// Mitsubishi GX Works2 project: SOFI_AmitGitai[1]   PLC: FX3G

// global labels: Global1
VAR_GLOBAL
  CreamTank AT D1102 : INT;
  ChocolateTank AT D1110 : INT;
  BiscuitTank AT D1106 : INT;
END_VAR
VAR_GLOBAL CONSTANT
  SUBCream : INT := 300;
  SUBBiscuit : INT := 6;
END_VAR
VAR_GLOBAL
  TurnON AT X010 : BOOL;
  InventoryDownload AT X011 : BOOL;
  EmergencyOff AT X005 : BOOL;
  ZilufOn AT Y004 : BOOL;
  Sen_15 AT X004 : BOOL;
  Ariza AT X000 : BOOL;
  Sen_camera AT X002 : BOOL;
  Sen_contact AT X003 : BOOL;
  MachineAOn AT M0 : BOOL;
  TCoil1 AT TC1 : BOOL;
  Light1 AT Y001 : BOOL;
  TS1change AT TS1 : BOOL;
  RestartTimer AT M1 : BOOL;
  TS2change AT TS2 : BOOL;
  Light0 AT Y000 : BOOL;
  TCoil2 AT TC2 : BOOL;
  TCoil0 AT TC0 : BOOL;
  TS0change AT TS0 : BOOL;
  StartDgima AT X006 : BOOL;
  analog_input_1 AT D8280 : INT;
  save_analog_value AT D8000 : INT;
  HelperLight2 AT M2 : BOOL;
  StartDay AT X007 : BOOL;
  StartLamp AT Y007 : BOOL;
  Sen_30 AT X001 : BOOL;
END_VAR
VAR_GLOBAL CONSTANT
  MinimumChocolate : INT := 240;
END_VAR
VAR_GLOBAL
  CreamInput AT D1100 : INT;
  ChocolateInput AT D1108 : INT;
  BiscuitInput AT D1104 : INT;
  TCoil3 AT TC3 : BOOL;
  TS3Hivhuv AT TS3 : BOOL;
  HelperGoodInventory AT M4 : BOOL;
END_VAR
VAR_GLOBAL CONSTANT
  TimerHivHuv1 : INT := 6;
  TimerHivHuv2 : INT := 6;
END_VAR
VAR_GLOBAL
  ZilufTank AT D1112 : INT;
END_VAR
VAR_GLOBAL CONSTANT
  Hivhuv : INT := 30;
  RegularCoating : INT := 5;
  ChocolateAmountCoating : INT := 120;
  DoubleCoatingMinimum : INT := 6;
  DoubleCoatimgMaximum : INT := 10;
END_VAR
VAR_GLOBAL
  CoatingLamp AT Y003 : BOOL;
  TvilaTank AT D1116 : INT;
END_VAR
VAR_GLOBAL CONSTANT
  ChocolateAmountCoating2 : INT := 240;
END_VAR
VAR_GLOBAL
  TCoil4 AT TC4 : BOOL;
END_VAR
VAR_GLOBAL CONSTANT
  Timer50 : INT := 50;
  TimerFor4seconds : INT := 40;
  normal_chocolate : INT := 400;
END_VAR
VAR_GLOBAL
  ChocolateInputCoating AT D1118 : INT;
  TS4ForLamp AT TS4 : BOOL;
END_VAR
VAR_GLOBAL CONSTANT
  ResetTvilaTank : INT;
END_VAR
VAR_GLOBAL
  OutputC AT CS1 : BOOL;
  ArizaLamp AT Y002 : BOOL;
  InputC2 AT CC2 : BOOL;
END_VAR
VAR_GLOBAL CONSTANT
  Counter6 : INT := 6;
  Counter5 : INT := 5;
END_VAR
VAR_GLOBAL
  OutputC2 AT CS2 : BOOL;
  InputC AT CC1 : BOOL;
  FinishInputReciever AT M13 : BOOL;
  KrembosAmount AT D1120 : INT;
END_VAR
VAR_GLOBAL CONSTANT
  MishtahFinish : INT := 6;
END_VAR
VAR_GLOBAL
  analog_output AT D8282 : INT;
  STAM AT Y011 : BOOL;
END_VAR
VAR_GLOBAL CONSTANT
  CONST : INT;
END_VAR
VAR_GLOBAL
  KremboNew AT D1121 : INT;
END_VAR
VAR_GLOBAL CONSTANT
  const10 : INT := 10;
  CONST400 : INT := 400;
  CONST40 : INT := 40;
END_VAR
VAR_GLOBAL
  SubIndication AT M6 : BOOL;
  DgimaLamp AT M9 : BOOL;
  HelperLight3 AT M3 : BOOL;
  NoInventory AT M5 : BOOL;
  RegularCoat AT M7 : BOOL;
  DoubleCoat AT M8 : BOOL;
  ChocolateSubInventory AT M10 : BOOL;
  FinishZiluf AT M11 : BOOL;
  HelperM12 AT M12 : BOOL;
  HelperM15 AT M15 : BOOL;
  HelperM14 AT M14 : BOOL;
  HelperM16 AT M16 : BOOL;
  HelperM17 AT M17 : BOOL;
  HelperM18 AT M18 : BOOL;
  HelperM19 AT M19 : BOOL;
  HelperM20 AT M20 : BOOL;
  HelperM21 AT M21 : BOOL;
  HelperM22 AT M22 : BOOL;
  GoodInventory AT M24 : BOOL;
  HelperM25 AT M25 : BOOL;
  HelperM26 AT M26 : BOOL;
  HelperM27 AT M27 : BOOL;
  FinishDay AT M28 : BOOL;
  HelperM23 AT M23 : BOOL;
  HelperM29 AT M29 : BOOL;
  TCoil5 AT TC5 : BOOL;
  TS5Reset AT TS5 : BOOL;
END_VAR

// task Task_01 (event TRUE, interval 0, priority 31): POU_01

PROGRAM POU_01
VAR
  TS4 : BOOL;
  TSForLamp : BOOL;
END_VAR
(* structured ladder/FBD written out as ST: instructions are called as NAME(EN, inputs, outputs); _pN, _eN, _tN stand for wires *)
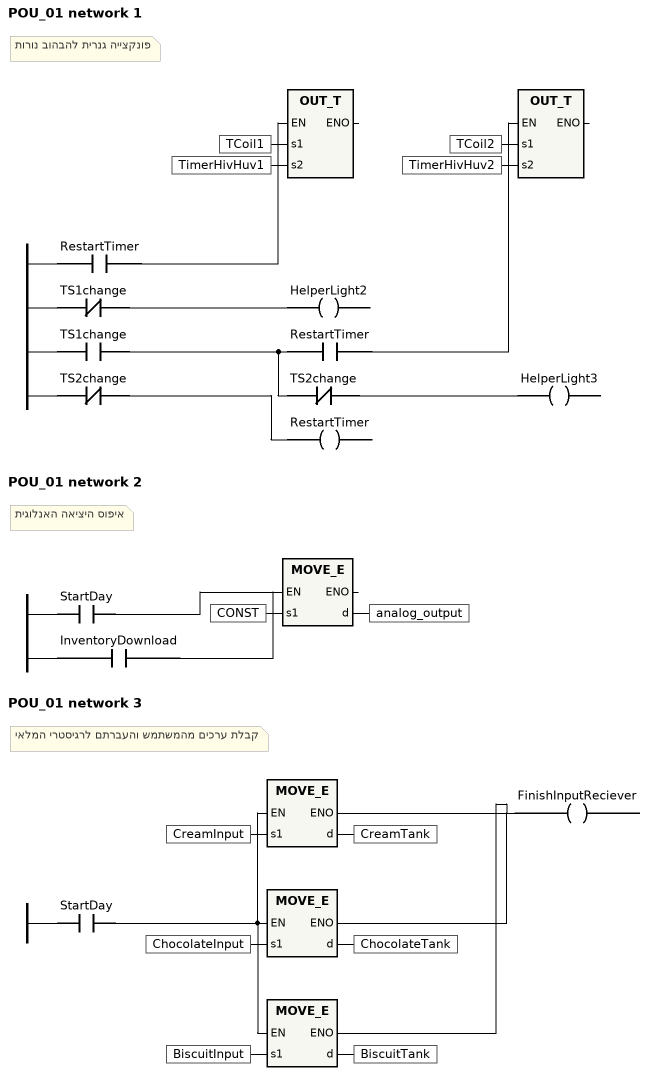
(* network 1 *)
(* פונקצייה גנרית להבהוב נורות *)
OUT_T(RestartTimer, TCoil1, TimerHivHuv1);
HelperLight2 := NOT TS1change;
OUT_T(TS1change AND RestartTimer, TCoil2, TimerHivHuv2);
HelperLight3 := TS1change AND NOT TS2change;
RestartTimer := NOT TS2change;
(* network 2 *)
(* איפוס היציאה האנלוגית *)
MOVE_E(StartDay OR InventoryDownload, CONST, analog_output);
(* network 3 *)
(* קבלת ערכים מהמשתמש והעברתם לרגיסטרי המלאי *)
_e1 := MOVE_E(StartDay, CreamInput, CreamTank);
_e2 := MOVE_E(StartDay, ChocolateInput, ChocolateTank);
_e3 := MOVE_E(StartDay, BiscuitInput, BiscuitTank);
FinishInputReciever := _e1 OR _e2 OR _e3;
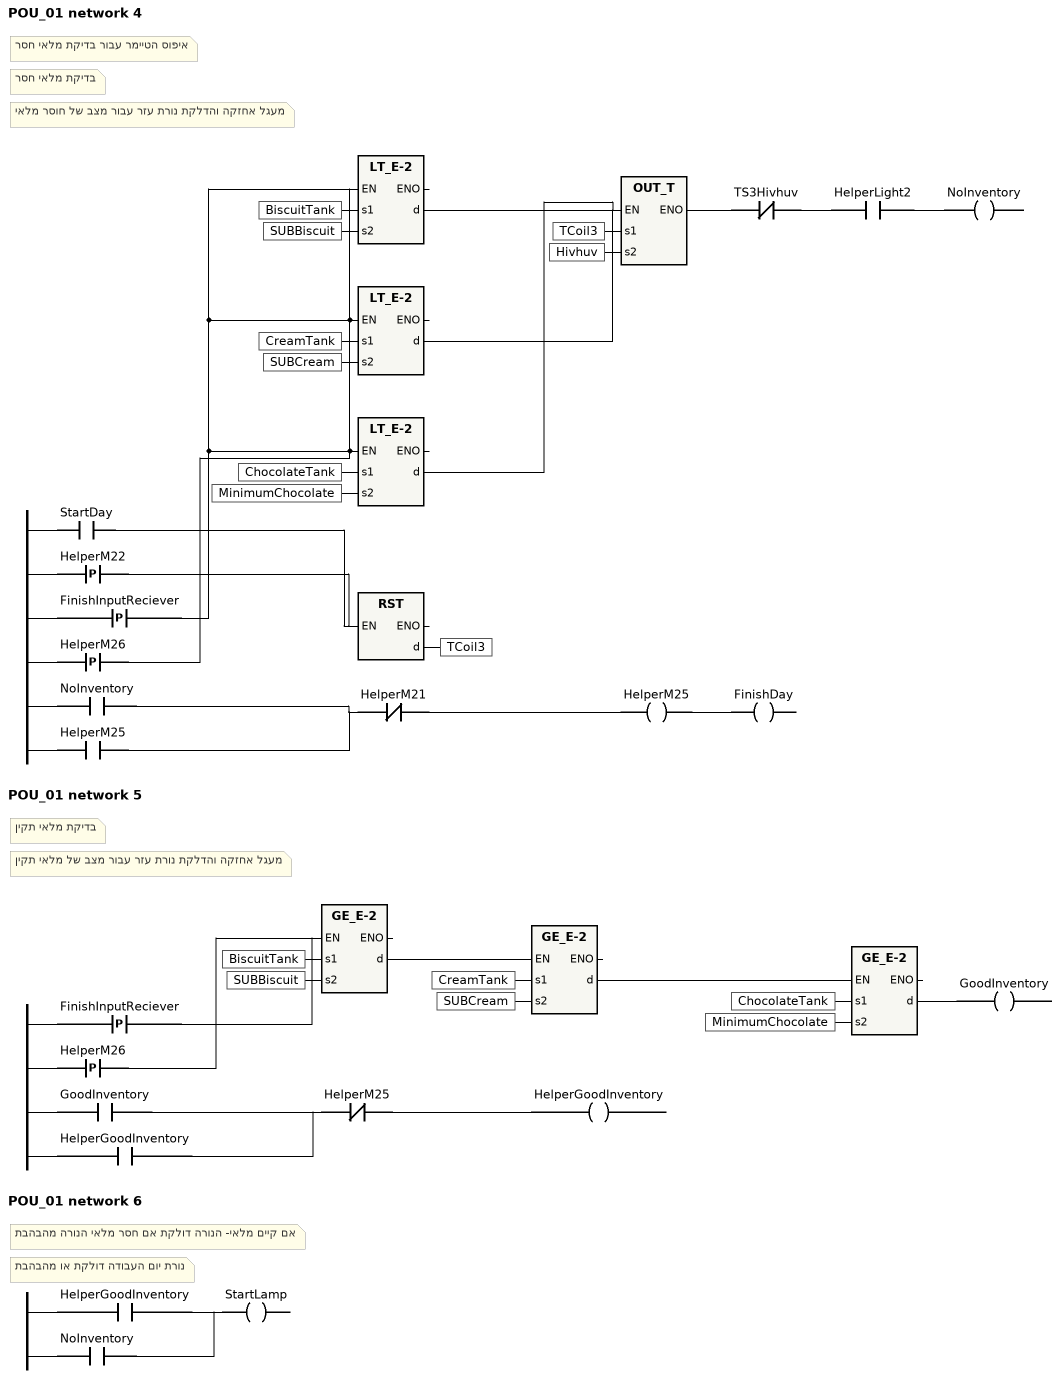
(* network 4 *)
(* איפוס הטיימר עבור בדיקת מלאי חסר *)
(* בדיקת מלאי חסר *)
(* מעגל אחזקה והדלקת נורת עזר עבור מצב של חוסר מלאי *)
RST(StartDay OR LDP(TRUE, HelperM22), TCoil3);
_p1 := LDP(TRUE, FinishInputReciever) OR LDP(TRUE, HelperM26);
LT_E(_p1, BiscuitTank, SUBBiscuit, _t2);
LT_E(_p1, CreamTank, SUBCream, _t3);
LT_E(_p1, ChocolateTank, MinimumChocolate, _t4);
_e5 := OUT_T(_t2 OR _t3 OR _t4, TCoil3, Hivhuv);
NoInventory := _e5 AND NOT TS3Hivhuv AND HelperLight2;
_p6 := (NoInventory OR HelperM25) AND NOT HelperM21;
HelperM25 := _p6;
FinishDay := _p6;
(* network 5 *)
(* בדיקת מלאי תקין *)
(* מעגל אחזקה והדלקת נורת עזר עבור מצב של מלאי תקין *)
GE_E(LDP(TRUE, FinishInputReciever) OR LDP(TRUE, HelperM26), BiscuitTank, SUBBiscuit, _t1);
GE_E(_t1, CreamTank, SUBCream, _t2);
GE_E(_t2, ChocolateTank, MinimumChocolate, _t3);
GoodInventory := _t3;
HelperGoodInventory := (GoodInventory OR HelperGoodInventory) AND NOT HelperM25;
(* network 6 *)
(* אם קיים מלאי- הנורה דולקת אם חסר מלאי הנורה מהבהבת *)
(* נורת יום העבודה דולקת או מהבהבת *)
StartLamp := HelperGoodInventory OR NoInventory;
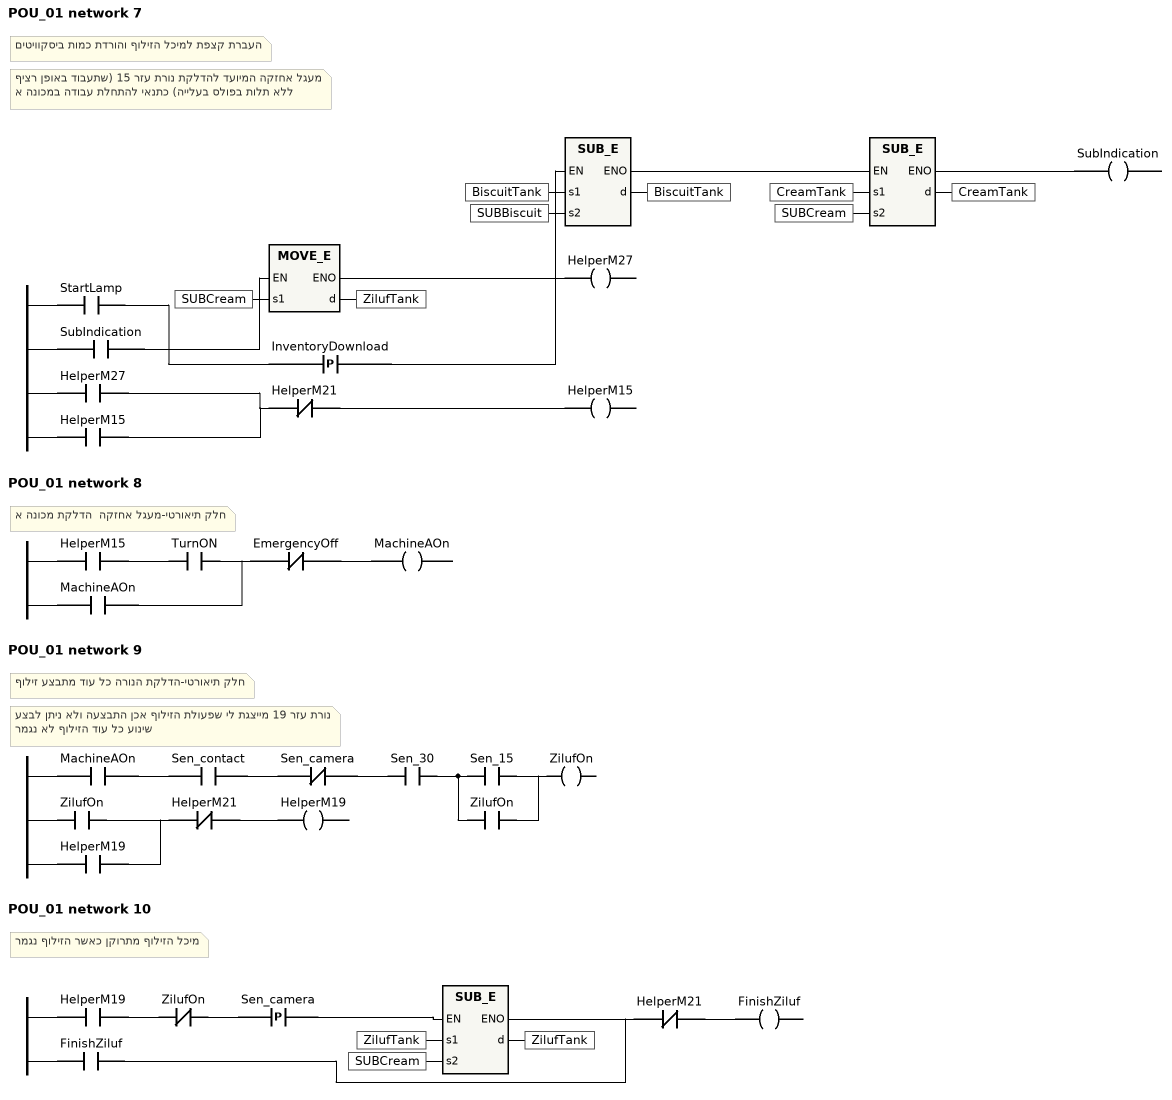
(* network 7 *)
(* העברת קצפת למיכל הזילוף והורדת כמות ביסקוויטים *)
(* מעגל אחזקה המיועד להדלקת נורת עזר 15 (שתעבוד באופן רציף ללא תלות בפולס בעלייה) כתנאי להתחלת עבודה במכונה א *)
_e1 := SUB_E(StartLamp AND LDP(TRUE, InventoryDownload), BiscuitTank, SUBBiscuit, BiscuitTank);
_e2 := SUB_E(_e1, CreamTank, SUBCream, CreamTank);
SubIndication := _e2;
_e3 := MOVE_E(SubIndication, SUBCream, ZilufTank);
HelperM27 := _e3;
HelperM15 := (HelperM27 OR HelperM15) AND NOT HelperM21;
(* network 8 *)
(* חלק תיאורטי-מעגל אחזקה  הדלקת מכונה א *)
MachineAOn := ((HelperM15 AND TurnON) OR MachineAOn) AND NOT EmergencyOff;
(* network 9 *)
(* חלק תיאורטי-הדלקת הנורה כל עוד מתבצע זילוף *)
(* נורת עזר 19 מייצגת לי שפעולת הזילוף אכן התבצעה ולא ניתן לבצע שינוע כל עוד הזילוף לא נגמר *)
_p1 := MachineAOn AND Sen_contact AND NOT Sen_camera AND Sen_30;
ZilufOn := (_p1 AND Sen_15) OR (_p1 AND ZilufOn);
HelperM19 := (ZilufOn OR HelperM19) AND NOT HelperM21;
(* network 10 *)
(* מיכל הזילוף מתרוקן כאשר הזילוף נגמר *)
_e1 := SUB_E(HelperM19 AND NOT ZilufOn AND LDP(TRUE, Sen_camera), ZilufTank, SUBCream, ZilufTank);
FinishZiluf := (_e1 OR FinishZiluf) AND NOT HelperM21;
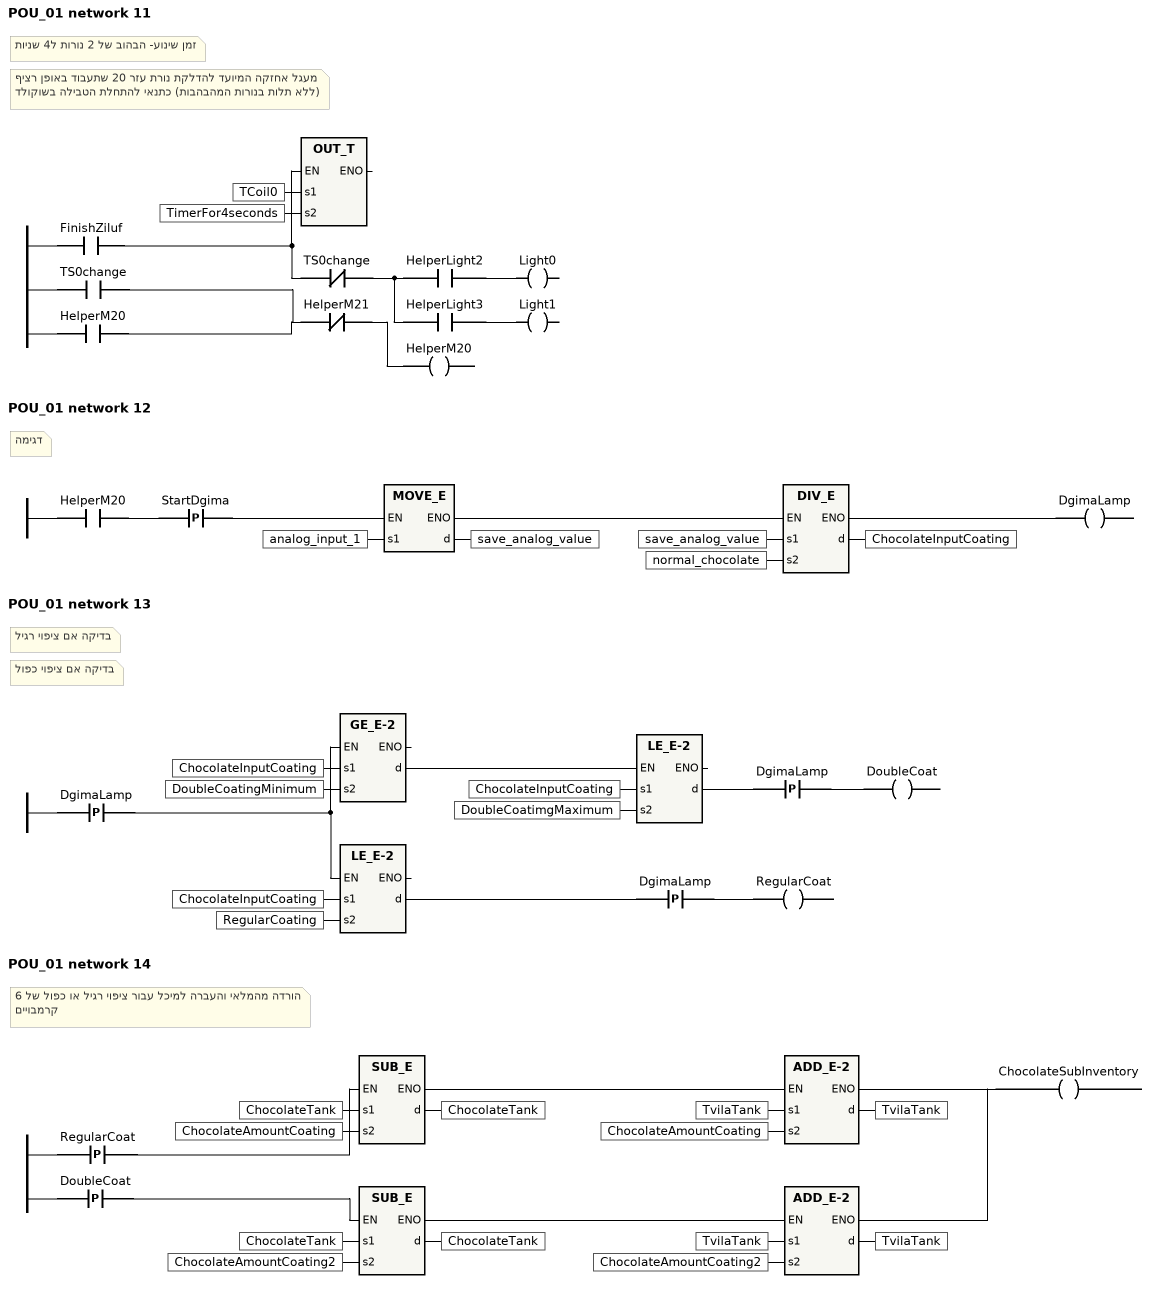
(* network 11 *)
(* זמן שינוע- הבהוב של 2 נורות ל4 שניות *)
(* מעגל אחזקה המיועד להדלקת נורת עזר 20 שתעבוד באופן רציף (ללא תלות בנורות המהבהבות) כתנאי להתחלת הטבילה בשוקולד *)
_p1 := FinishZiluf AND NOT TS0change;
Light0 := _p1 AND HelperLight2;
OUT_T(FinishZiluf, TCoil0, TimerFor4seconds);
Light1 := _p1 AND HelperLight3;
HelperM20 := (TS0change OR HelperM20) AND NOT HelperM21;
(* network 12 *)
(* דגימה *)
_e1 := MOVE_E(HelperM20 AND LDP(TRUE, StartDgima), analog_input_1, save_analog_value);
_e2 := DIV_E(_e1, save_analog_value, normal_chocolate, ChocolateInputCoating);
DgimaLamp := _e2;
(* network 13 *)
(* בדיקה אם ציפוי רגיל *)
(* בדיקה אם ציפוי כפול *)
_p1 := LDP(TRUE, DgimaLamp);
LE_E(_p1, ChocolateInputCoating, RegularCoating, _t2);
RegularCoat := _t2 AND LDP(TRUE, DgimaLamp);
GE_E(_p1, ChocolateInputCoating, DoubleCoatingMinimum, _t3);
LE_E(_t3, ChocolateInputCoating, DoubleCoatimgMaximum, _t4);
DoubleCoat := _t4 AND LDP(TRUE, DgimaLamp);
(* network 14 *)
(* הורדה מהמלאי והעברה למיכל עבור ציפוי רגיל או כפול של 6 קרמבויים *)
_e1 := SUB_E(LDP(TRUE, RegularCoat), ChocolateTank, ChocolateAmountCoating, ChocolateTank);
_e2 := ADD_E(_e1, TvilaTank, ChocolateAmountCoating, TvilaTank);
_e3 := SUB_E(LDP(TRUE, DoubleCoat), ChocolateTank, ChocolateAmountCoating2, ChocolateTank);
_e4 := ADD_E(_e3, TvilaTank, ChocolateAmountCoating2, TvilaTank);
ChocolateSubInventory := _e2 OR _e4;
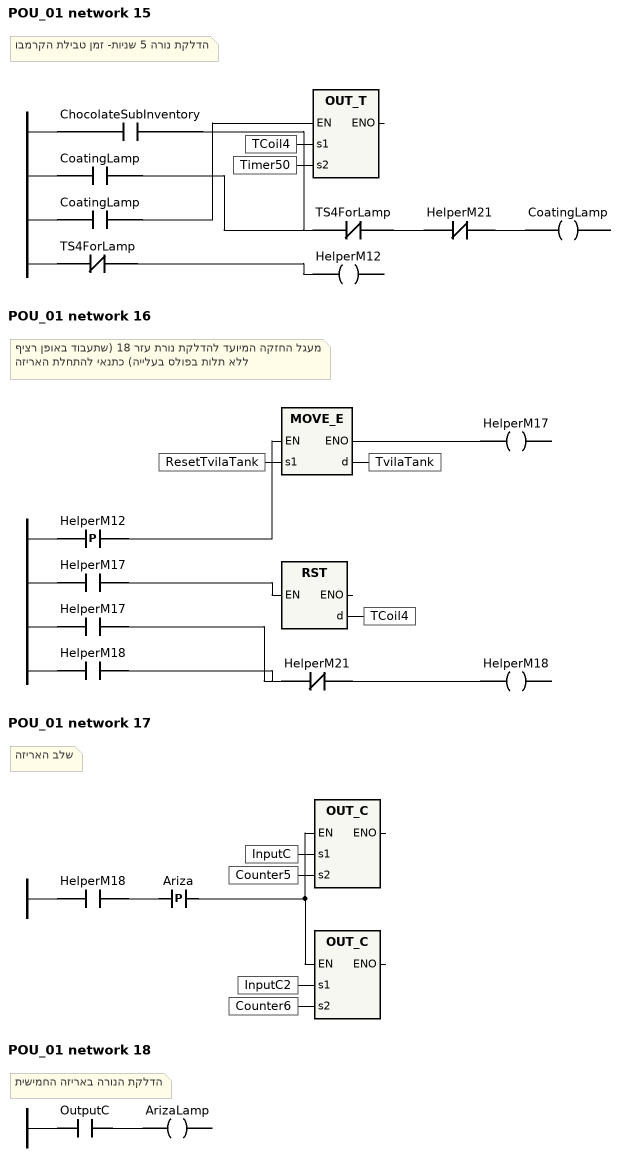
(* network 15 *)
(* הדלקת נורה 5 שניות- זמן טבילת הקרמבו *)
CoatingLamp := ((ChocolateSubInventory OR CoatingLamp) AND NOT TS4ForLamp) AND NOT HelperM21;
OUT_T(CoatingLamp, TCoil4, Timer50);
HelperM12 := NOT TS4ForLamp;
(* network 16 *)
(* מעגל החזקה המיועד להדלקת נורת עזר 18 (שתעבוד באופן רציף ללא תלות בפולס בעלייה) כתנאי להתחלת האריזה *)
_e1 := MOVE_E(LDP(TRUE, HelperM12), ResetTvilaTank, TvilaTank);
HelperM17 := _e1;
RST(HelperM17, TCoil4);
HelperM18 := (HelperM17 OR HelperM18) AND NOT HelperM21;
(* network 17 *)
(* שלב האריזה *)
_p1 := HelperM18 AND LDP(TRUE, Ariza);
OUT_C(_p1, InputC, Counter5);
OUT_C(_p1, InputC2, Counter6);
(* network 18 *)
(* הדלקת הנורה באריזה החמישית *)
ArizaLamp := OutputC;
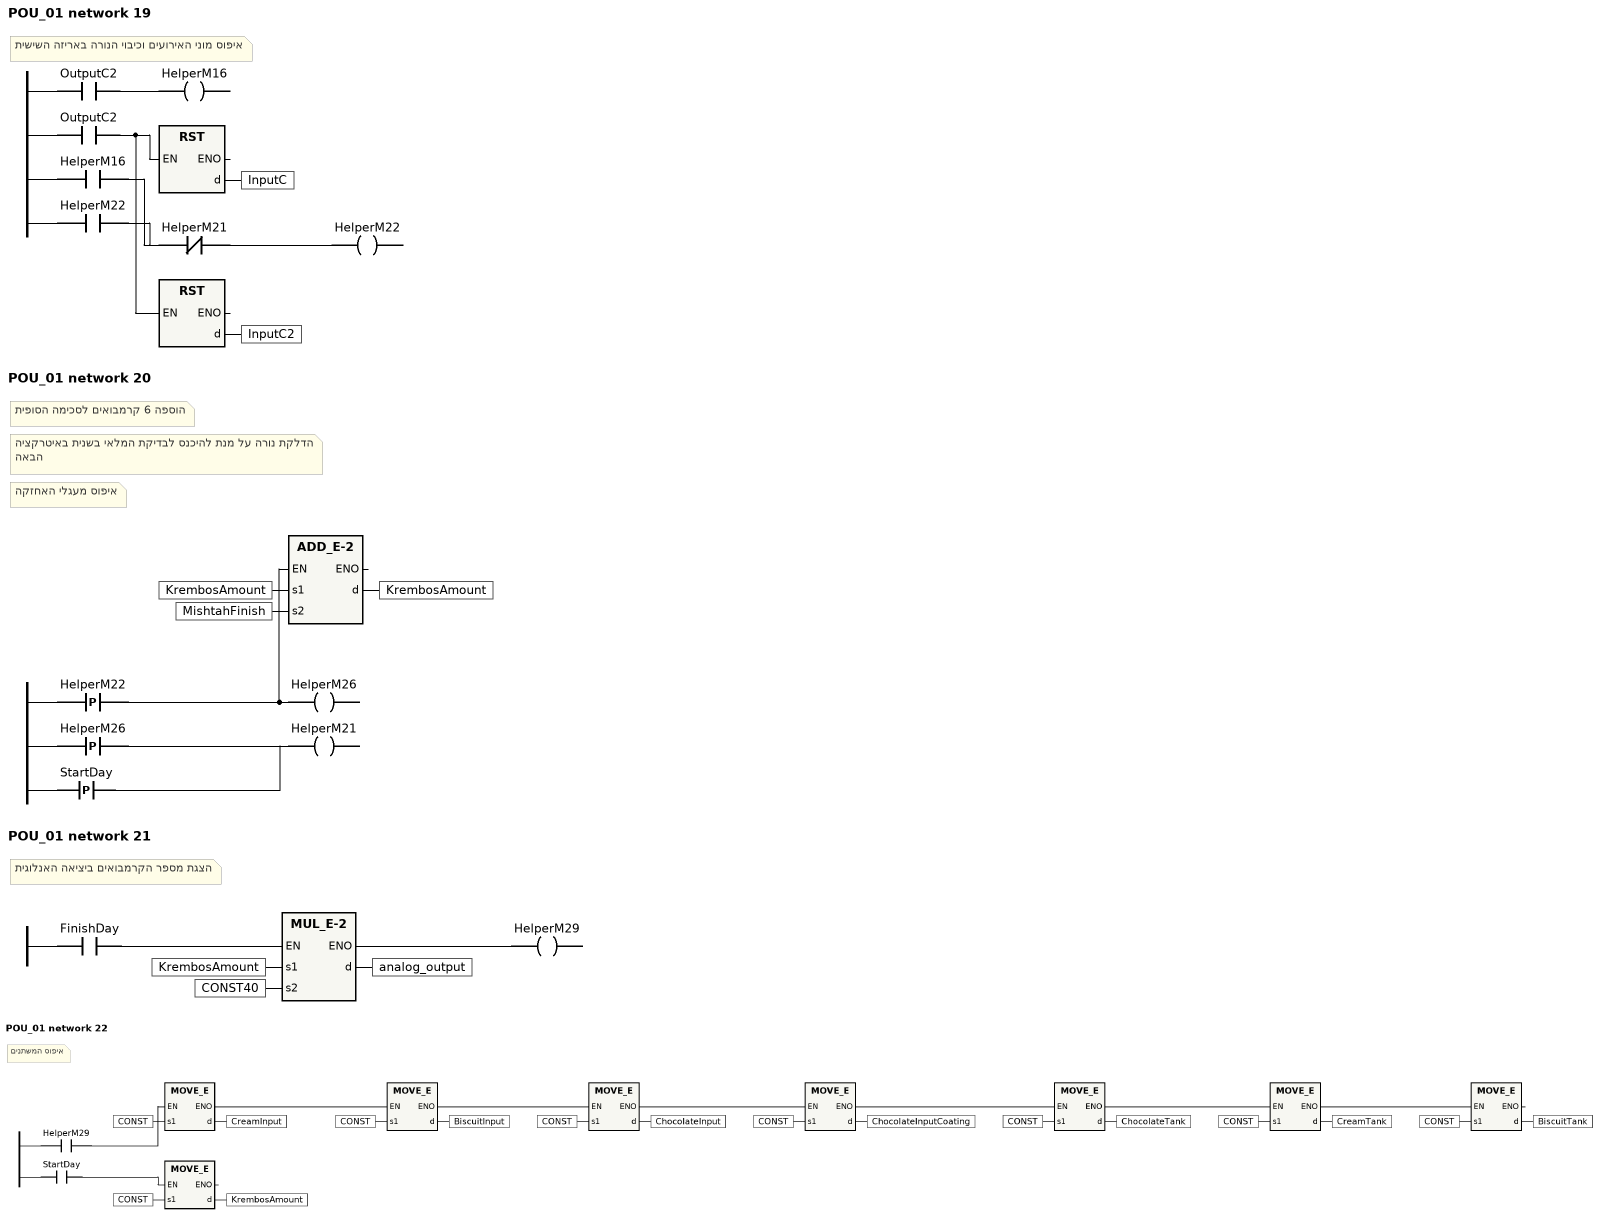
(* network 19 *)
(* איפוס מוני האירועים וכיבוי הנורה באריזה השישית *)
HelperM16 := OutputC2;
RST(OutputC2, InputC);
RST(OutputC2, InputC2);
HelperM22 := (HelperM16 OR HelperM22) AND NOT HelperM21;
(* network 20 *)
(* הוספה 6 קרמבואים לסכימה הסופית *)
(* הדלקת נורה על מנת להיכנס לבדיקת המלאי בשנית באיטרקציה הבאה *)
(* איפוס מעגלי האחזקה *)
_p1 := LDP(TRUE, HelperM22);
ADD_E(_p1, KrembosAmount, MishtahFinish, KrembosAmount);
HelperM26 := _p1;
HelperM21 := LDP(TRUE, HelperM26) OR LDP(TRUE, StartDay);
(* network 21 *)
(* הצגת מספר הקרמבואים ביציאה האנלוגית *)
_e1 := MUL_E(FinishDay, KrembosAmount, CONST40, analog_output);
HelperM29 := _e1;
(* network 22 *)
(* איפוס המשתנים *)
_e1 := MOVE_E(HelperM29, CONST, CreamInput);
_e2 := MOVE_E(_e1, CONST, BiscuitInput);
_e3 := MOVE_E(_e2, CONST, ChocolateInput);
_e4 := MOVE_E(_e3, CONST, ChocolateInputCoating);
_e5 := MOVE_E(_e4, CONST, ChocolateTank);
_e6 := MOVE_E(_e5, CONST, CreamTank);
MOVE_E(_e6, CONST, BiscuitTank);
MOVE_E(StartDay, CONST, KrembosAmount);
END_PROGRAM
